// TIA Portal V21 export
FUNCTION_BLOCK "GestWatchdog_Bit"   // FB9, LAD
{ S7_Optimized_Access := 'TRUE' }
// stored: MemoryReserve 100, SetENOAutomatically false
   VAR_INPUT
      Watchdog_Recive : Bool;
      Reset : Bool;
   END_VAR
   VAR_OUTPUT
      Watchdog_Send : Bool;
   END_VAR
   VAR_IN_OUT
      Allarme : Bool;
   END_VAR
   VAR
      Watchdog_Prec : Bool;
      TimerAllarme : "Std_stTimer";
   END_VAR
BEGIN

REGION Network 1
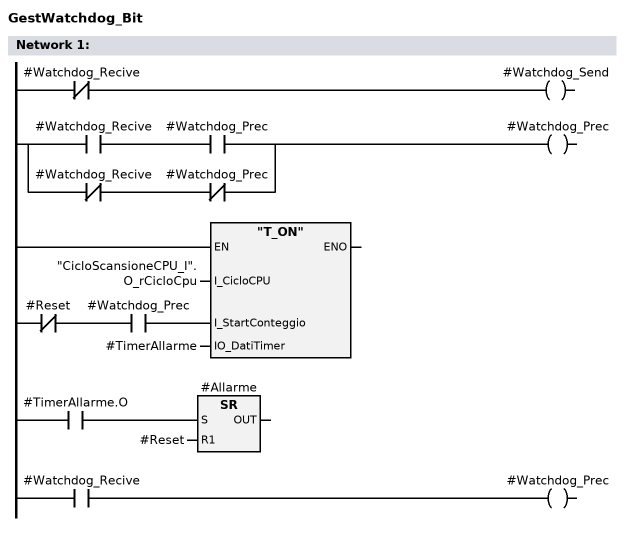
   RUNG wire#powerrail
      I_Contact( #Watchdog_Recive )
      Coil( #Watchdog_Send )
   END_RUNG
   RUNG wire#powerrail
      Contact( #Watchdog_Recive )
      Contact( #Watchdog_Prec )
      wire#w1
      Coil( #Watchdog_Prec )
   END_RUNG
   RUNG wire#powerrail
      I_Contact( #Watchdog_Recive )
      I_Contact( #Watchdog_Prec )
   END_RUNG wire#w1
   RUNG wire#powerrail
      "T_ON"(I_StartConteggio := wire#w2, I_CicloCPU := "CicloScansioneCPU_I".O_rCicloCpu, IO_DatiTimer := #TimerAllarme)
   END_RUNG
   RUNG wire#powerrail
      I_Contact( #Reset )
      Contact( #Watchdog_Prec )
   END_RUNG wire#w2
   RUNG wire#powerrail
      Contact( #TimerAllarme.O )
      S_SR(operand := #Allarme, r1 := #Reset)
   END_RUNG
   RUNG wire#powerrail
      Contact( #Watchdog_Recive )
      Coil( #Watchdog_Prec )
   END_RUNG
   // the same network as SCL:
   #Watchdog_Send := NOT #Watchdog_Recive;
   #Watchdog_Prec := (#Watchdog_Recive AND #Watchdog_Prec) OR (NOT #Watchdog_Recive AND NOT #Watchdog_Prec);
   "T_ON"(I_CicloCPU := "CicloScansioneCPU_I".O_rCicloCpu,
          I_StartConteggio := NOT #Reset AND #Watchdog_Prec,
          IO_DatiTimer := #TimerAllarme);
   IF #TimerAllarme.O THEN
       #Allarme := TRUE;   // SR flip-flop
   END_IF;
   IF #Reset THEN #Allarme := FALSE; END_IF;
   #Watchdog_Prec := #Watchdog_Recive;
END_REGION

REGION Network 2 (SCL)
   #TimerAllarme.Preset := 6.0;
END_REGION
END_FUNCTION_BLOCK
